{attribute 'qualified_only'}
{attribute 'strict'}
{attribute 'to_string'}
TYPE FILE_LOGGER_STATE_MACHINE :
(
	INITIAL, 
	LOGGING, 
	FAILED
);
END_TYPE

(* stored: Version 1.1.0.1
   DUT FILE_LOGGER_STATE_MACHINE: Id {b0a8aecb-720a-45ce-a1f2-2acb5d93911d} *)
